// TIA Portal project "LQG" (V16)
// Vorlageprojekt für das Buch mit Zielsystem S7-1200

(* hardware
DEVICE "S7-1200-Station_1"  S7-1200 Station
   slot 0: "Baugruppenträger_0"  Rack  V1.0
   slot 1: "PLC_1"  CPU 1211C DC/DC/DC  6ES7 211-1AE40-0XB0  V4.1
   slot 3: "AQ 1x12BIT_1"  AQ1 signal board  6ES7 232-4HA30-0XB0  V1.0
DEVICE "HMI_1"  TP900 Comfort
   slot 0: "HMI_1"  TP900 Comfort  6AV2 124-0JC01-0AX0  16.0.0.0
   slot 1: "HMI_RT_1"  TP900 Comfort  6AV2 124-0JC01-0AX0  16.0.0.0
   slot 5: "HMI_1.IE_CP_1"  PROFINET Interface  16.0.0.0
      slot 1: "Interfaz PROFINET_1"  PROFINET Interface
         slot 1: "Port_1"  Port
         slot 2: "Port_2"  Port
   slot 7: "HMI_1.MPI/DP_CP_1"  MPI/DP Interface  16.0.0.0
*)

// ===== PLC "PLC_1"  CPU 1211C DC/DC/DC =====

VAR_GLOBAL   // PLC tag table "Standard-Variablentabelle"
   "l2" AT %MD40 : Real;
   "l1" AT %MD44 : Real;
   "Kd1" AT %MD0 : Real;
   "Kd2" AT %MD4 : Real;
   "x1e" AT %MD8 : Real;
   "x2e" AT %MD12 : Real;
   "ue" AT %MD16 : Real;
   "u_min" AT %MD20 : Real;
   "u_max" AT %MD24 : Real;
   "z1" AT %MD28 : Real;
   "z2" AT %MD32 : Real;
   "delta_u" AT %MD36 : Real;
   "u_out" AT %MD48 : Real;
   "v1" AT %QD4 : Real;
   "AI_L1" AT %ID4 : Real;
   "AI_L2" AT %ID8 : Real;
   "AO_u" AT %QD0 : Real;
   "FLOWMETER1" AT %ID12 : Real;
   "FLOWMETER2" AT %ID16 : Real;
   "DISCHARGE1" AT %QD8 : Real;
   "DISCHARGE2" AT %QD12 : Real;
   "x1_hat" AT %MD52 : Real;
   "x2_hat" AT %MD56 : Real;
   "L1_1" AT %MD60 : Real;
   "L1_2" AT %MD64 : Real;
   "L2_1" AT %MD68 : Real;
   "L2_2" AT %MD72 : Real;
   "y1_dev" AT %MD76 : Real;
   "y2_dev" AT %MD80 : Real;
   "x1_hat_dev" AT %MD84 : Real;
   "x2_hat_dev" AT %MD88 : Real;
   "corr1" AT %MD92 : Real;
   "corr2" AT %MD96 : Real;
   "A11" AT %MD100 : Real;
   "A12" AT %MD104 : Real;
   "A21" AT %MD108 : Real;
   "A22" AT %MD112 : Real;
   "B1" AT %MD116 : Real;
   "B2" AT %MD120 : Real;
   "resid1" AT %MD124 : Real;
   "resid2" AT %MD128 : Real;
   "pred1" AT %MD132 : Real;
   "pred2" AT %MD136 : Real;
   "corr_term1" AT %MD140 : Real;
   "corr_term2" AT %MD144 : Real;
   "disp" AT %QD16 : Real;
   "err1" AT %MD148 : Real;
   "err2" AT %MD152 : Real;
   "start" AT %I30.0 : Bool;
   "lqg11" AT %Q62.0 : Bool;
   "lqg22" AT %Q62.1 : Bool;
   "statSeed" AT %MD156 : DInt;
   "noise1" AT %MD160 : Real;
   "noise2" AT %MD164 : Real;
   "l1_ruido" AT %MD168 : Real;
   "l2_ruido" AT %MD172 : Real;
END_VAR

DATA_BLOCK "OnOff_DB"   // DB2
{ S7_Optimized_Access := 'TRUE' }
VERSION : 0.1
// stored: InstanceOfName OnOff
"OnOff"
BEGIN
END_DATA_BLOCK

DATA_BLOCK "OnOff_DB2"   // DB4
{ S7_Optimized_Access := 'TRUE' }
VERSION : 0.1
// stored: InstanceOfName OnOff
"OnOff"
BEGIN
END_DATA_BLOCK

DATA_BLOCK "OnOff_DB_1"   // DB5
{ S7_Optimized_Access := 'TRUE' }
VERSION : 0.1
// stored: InstanceOfName OnOff
"OnOff"
BEGIN
END_DATA_BLOCK

DATA_BLOCK "I"   // DB6
{ S7_Optimized_Access := 'TRUE' }
VERSION : 0.1
// stored: InstanceOfName lqg1
"lqg1"
BEGIN
END_DATA_BLOCK

FUNCTION_BLOCK "OnOff"   // FB1, SCL
{ S7_Optimized_Access := 'TRUE' }
VERSION : 0.1
BEGIN
   // ==============================
   // PARÁMETROS EXISTENTES (NO TOCAR)
   // ==============================
   "DISCHARGE1" := 4.5;
   "DISCHARGE2" := 5;
   "A11" := -0.010796;
   "A12" := 0.0132014;
   "A21" := 0.0;
   "A22" := -0.01320;

   "B1" := 0.0;
   "B2" := 0.007957;

   "Kd1" := 24.302648160374716;
   "Kd2" := 7.403861999025946;

   "x1e" := 2.0000;
   "x2e" := 1.6357;
   "ue" := 5.2091; ///////////

   "u_min" := 0.0;
   "u_max" := 10.0;

   // ==============================
   // 1) SENSOR SIN CALIBRACIÓN
   // ==============================

   "l1" := "AI_L1" * 0.3;
   "l2" := "AI_L2" * 0.3;
   "v1" := 4.073 * SQRT("AI_L2" * 0.3);
   // ==============================
   // 2) MATRIZ L DEL KALMAN
   // ==============================

   "L1_1" := 31.612416940708904;
   "L1_2" := 0.006333174290898;
   "L2_1" := 0.006333174290897;
   "L2_2" := 31.610107079825518;

   // ==============================
   // 3) CÁLCULOS PREVIOS
   // ==============================

   // Desviaciones de los sensores (Real)

   "y1_dev" := "l1" - "x1e";
   "y2_dev" := "l2" - "x2e";


   // Desviaciones del Estimado (Anterior)

   "x1_hat_dev" := "x1_hat" - "x1e";
   "x2_hat_dev" := "x2_hat" - "x2e";


   // Cálculo del Control LQR (basado en el estado estimado actual)
   "delta_u" := - ("Kd1" * "x1_hat_dev" + "Kd2" * "x2_hat_dev");

   // ==============================
   // 4) OBSERVADOR DE KALMAN (CORREGIDO)
   // ==============================

   // Error de estimación (Medición - Estimación)
   // Usamos variables temporales para no confundirnos

   "err1" := "y1_dev" - "x1_hat_dev";
   "err2" := "y2_dev" - "x2_hat_dev";

   // CÁLCULO DE LA DERIVADA (corr = Ax + Bu + L*error)
   // Aquí estaba el problema antes. Esta es la forma segura:

   "corr1" := ("A11" * "x1_hat_dev") + ("A12" * "x2_hat_dev")

   + ("B1" * "delta_u")

   + ("L1_1" * "err1") + ("L1_2" * "err2");



   "corr2" := ("A21" * "x1_hat_dev") + ("A22" * "x2_hat_dev")

   + ("B2" * "delta_u")

   + ("L2_1" * "err1") + ("L2_2" * "err2");



   // INTEGRACIÓN (ACTUALIZAR ESTADOS)

   // IMPORTANTE: Solo se hace UNA vez y con 0.05 (no 0.5)

   "x1_hat" := "x1_hat" + 0.05 * "corr1";

   "x2_hat" := "x2_hat" + 0.05 * "corr2";



   // Visualización para debug

   "disp" := "x1_hat_dev";



   // ==============================

   // 5) SEÑAL TOTAL Y SATURACIÓN

   // ==============================



   "u_out" := "ue" + "delta_u";



   IF "u_out" > "u_max" THEN



       "u_out" := "u_max";

   ELSIF "u_out" < "u_min" THEN



       "u_out" := "u_min";

   END_IF;



   // ==============================

   // 7) SALIDA AL ACTUADOR

   // ==============================

   "AO_u" := "u_out";



   // ==============================

   // EXTRA: TU CAUDAL

   // ==============================
END_FUNCTION_BLOCK

FUNCTION_BLOCK "lqg1"   // FB2, SCL
{ S7_Optimized_Access := 'TRUE' }
VERSION : 0.1
BEGIN
   // ==============================
   // GENERACIÓN DE RUIDO (SIMULACIÓN)
   // ==============================
   // Usamos DINT para el cálculo de la semilla y evitamos operadores lógicos
   "statSeed" := ("statSeed" * 1103515245 + 12345);

   // Aseguramos que sea positivo para la división (Absoluto manual)
   IF "statSeed" < 0 THEN
       "statSeed" := "statSeed" * -1;
   END_IF;

   // noise                                                      change
   "noise1" := ((DINT_TO_REAL("statSeed") / 2147483647.0) - 0.5) * 0;
   "noise2" := ((DINT_TO_REAL("statSeed") / 2147483647.0) - 0.5) * 0;

   // ==============================
   // PARÁMETROS EXISTENTES (NO TOCAR)
   // ==============================
   "DISCHARGE1" := 4.5;
   "DISCHARGE2" := 5;
   "A11" := -0.010796;
   "A12" := 0.0132014;
   "A21" := 0.0;
   "A22" := -0.01320;

   "B1" := 0.0;
   "B2" := 0.007957;

   "Kd1" := 23.824873879011026;
   "Kd2" := 7.752628045467919;

   "x1e" := 1.5000;
   "x2e" := 1.2268;
   "ue" := 4.5113;

   "u_min" := 0.00;
   "u_max" := 10.0;

   // ==============================
   // 1) SENSOR Y SIMULACIÓN DE RUIDO
   // ==============================

   "l1" := "AI_L1" * 0.3;
   "l2" := "AI_L2" * 0.3;

   // Variables con ruido para el observador
   "l1_ruido" := "l1" + "noise1";
   "l2_ruido" := "l2" + "noise2";

   "v1" := 4.073 * SQRT("l2_ruido");

   // ==============================
   // 2) MATRIZ L DEL KALMAN
   // ==============================

   "L1_1" := 9.988042526909684;
   "L1_2" := 0.013098451274169;
   "L2_1" := 0.000130984512741;
   "L2_2" := 0.985474476955653;

   // ==============================
   // 3) CÁLCULOS PREVIOS
   // ==============================

   // Desviaciones de los sensores (Usando l1_ruido y l2_ruido)
   "y1_dev" := "l1_ruido" - "x1e";
   "y2_dev" := "l2_ruido" - "x2e";

   // Desviaciones del Estimado (Anterior)
   "x1_hat_dev" := "x1_hat" - "x1e";
   "x2_hat_dev" := "x2_hat" - "x2e";

   // Cálculo del Control LQR (basado en el estado estimado actual)
   "delta_u" := - ("Kd1" * "x1_hat_dev" + "Kd2" * "x2_hat_dev");

   // ==============================
   // 4) OBSERVADOR DE KALMAN (CORREGIDO)
   // ==============================

   // Error de estimación (Medición con ruido - Estimación)
   "err1" := "y1_dev" - "x1_hat_dev";
   "err2" := "y2_dev" - "x2_hat_dev";

   // CÁLCULO DE LA DERIVADA (corr = Ax + Bu + L*error)
   "corr1" := ("A11" * "x1_hat_dev") + ("A12" * "x2_hat_dev")
   + ("B1" * "delta_u")
   + ("L1_1" * "err1") + ("L1_2" * "err2");

   "corr2" := ("A21" * "x1_hat_dev") + ("A22" * "x2_hat_dev")
   + ("B2" * "delta_u")
   + ("L2_1" * "err1") + ("L2_2" * "err2");

   // INTEGRACIÓN (Típicamente cada 50ms)
   "x1_hat" := "x1_hat" + 0.05 * "corr1";
   "x2_hat" := "x2_hat" + 0.05 * "corr2";

   // Visualización para debug
   "disp" := "x1_hat_dev";

   // ==============================
   // 5) SEÑAL TOTAL Y SATURACIÓN
   // ==============================

   "u_out" := "ue" + "delta_u";

   IF "u_out" > "u_max" THEN
       "u_out" := "u_max";
   ELSIF "u_out" < "u_min" THEN
       "u_out" := "u_min";
   END_IF;

   // ==============================
   // 7) SALIDA AL ACTUADOR
   // ==============================

   "AO_u" := 5;
END_FUNCTION_BLOCK

FUNCTION "MHJ-PLC-Lab-Function-S71200" : Void   // FC9000, SCL
{ S7_Optimized_Access := 'TRUE' }
VERSION : 0.1
   VAR_TEMP
      rdTimeReturn : Int;
      outputTime : DTL;
      SyncVal : Byte;
      forVal : Int;
      forVal_2 : Int;
      Value : Byte;
   END_VAR
   VAR CONSTANT
      CompVal : Byte := 16#34;
      Value_01 : Byte := 16#11;
      Value_01_DW : DWord := 16#A165_D992;
      Value_02_DW : DWord := 16#58BE_4401;
   END_VAR
BEGIN

   #Value:=PEEK(area := 16#82,
        dbNumber := 0,
        byteOffset := 511);
   #Value := #Value + 1;

   POKE(area := 16#82,
        dbNumber := 0,
        byteOffset := 511,
        value := #Value);

   POKE(area:=16#81,
        dbNumber:=0,
        byteOffset:=1016,
        value:=#Value_01_DW);
   POKE(area := 16#81,
        dbNumber := 0,
        byteOffset := 1020,
        value := #Value_02_DW);

   POKE(area := 16#81,
        dbNumber := 0,
        byteOffset := 511,
        value := B#16#00);

   FOR #forVal := 0 TO 120 DO
       FOR #forVal_2:=0 TO 10 DO
           #rdTimeReturn:=RD_SYS_T(#outputTime);
           #rdTimeReturn := WR_SYS_T(#outputTime);
           #rdTimeReturn := RD_SYS_T(#outputTime);
           #rdTimeReturn := WR_SYS_T(#outputTime);
       END_FOR;
       #SyncVal:= PEEK(area := 16#81,
                      dbNumber := 0,
                      byteOffset := 511);
       IF #SyncVal = #CompVal THEN
          GOTO M_1;
       END_IF;
   END_FOR;
   RETURN;

   M_1:
   POKE(area := 16#81,
        dbNumber := 0,
        byteOffset := 511,
        value := B#16#0);
END_FUNCTION

ORGANIZATION_BLOCK "Main"   // OB1, LAD, ProgramCycle
TITLE = "Main Program Sweep (Cycle)"
{ S7_Optimized_Access := 'TRUE' }
VERSION : 0.1
   VAR_INPUT
      Initial_Call : Bool;   // Initial call of this OB
      Remanence : Bool;   // =True, if remanent data are available
   END_VAR
BEGIN

REGION Network 1: Konnektierungsbaustein für PLC-Lab
   // Im Netzwerk 1 wird der Konnektierungsbaustein für PLC-Lab aufgerufen.
   // Dieser Aufruf darf nicht entfernt werden!
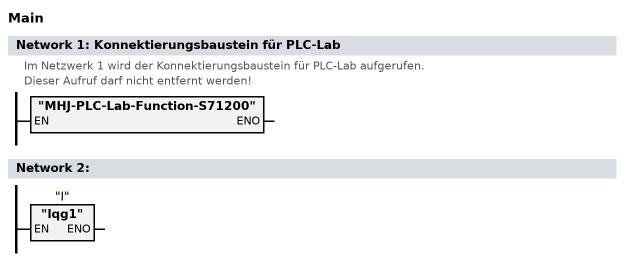
   RUNG wire#powerrail
      "MHJ-PLC-Lab-Function-S71200"()
   END_RUNG
   // the same network as SCL:
   "MHJ-PLC-Lab-Function-S71200"();
END_REGION

REGION Network 2
   RUNG wire#powerrail
      "I"()
   END_RUNG
   // the same network as SCL:
   "I"();   // "lqg1"
END_REGION
END_ORGANIZATION_BLOCK

(* ===== HMI "HMI_RT_1" =====
system functions are stored by id; their names below are inferred from use
connection "HMI_Conexión_1": ETHERNET, S7_1200_OMS

HMI tags "Tabla de variables estándar"
   "Número_imagen_variable" : UInt, internal
   "l1" : Real = PLC l1 AT %MD44, 1 s
   "l2" : Real = PLC l2 AT %MD40, 1 s
   "AO_u" : Real = PLC AO_u AT %QD0, 1 s

screen "Imagen raíz" 800x420, template "Plantilla_1"
   on GenerateScreen: SetTag("Número_imagen_variable", 1)
   TrendView "Visor de curvas_1" at 8,5 size 787x351

Template "Plantilla_1" 800x420
   Button "Exit" at 720,360 size 78x58; TextOff 'Exit'; PictureOff "ExitRuntime_TP900_Comfort_TR"; PictureOn "ExitRuntime_TP900_Comfort_TR"
      on Release: StopRuntime(0)
   Button "Template_Button" at 640,360 size 78x58; TextOff 'Text'
   Button "Template_Button_1" at 560,360 size 78x58; TextOff 'Text'
   Button "Template_Button_2" at 480,360 size 78x58; TextOff 'Text'
   Button "Template_Button_3" at 400,360 size 78x58; TextOff 'Text'
   Button "Template_Button_4" at 321,360 size 78x58; TextOff 'Text'
   Button "Template_Button_5" at 241,360 size 78x58; TextOff 'Text'
   Button "Template_Button_6" at 161,360 size 78x58; TextOff 'Text'
   Button "Template_Button_7" at 81,360 size 78x58; TextOff 'Text'
   Button "Start screen" at 1,360 size 78x58; TextOff 'Start screen'; PictureOff "NavigateHome_TP900_Comfort_TR"; PictureOn "NavigateHome_TP900_Comfort_TR"
      on Release: ActivateScreen("Imagen raíz", 0)
*)